FUNCTION_BLOCK TimerServer (* Updates time upon every REQ event and can be used to request time remotely. *)
  (* Standard: 61499-2 *)
  (* Version 1.0, 2017-09-05, Marc Jakobi, HTW Berlin *)
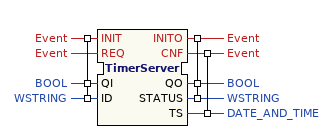
  EVENT_INPUT
    INIT WITH QI, ID; (* Initialization Request *)
    REQ; (* Service Request Event *)
  END_EVENT
  EVENT_OUTPUT
    INITO WITH QO, STATUS; (* Initialization Confirm *)
    CNF WITH TS; (* Service Indication *)
  END_EVENT
  VAR_INPUT
    QI : BOOL; (* Input event qualifier *)
    ID : WSTRING; (* Connection identifier *)
  END_VAR
  VAR_OUTPUT
    QO : BOOL; (* Output event qualifier *)
    STATUS : WSTRING; (* Service status *)
    TS : DATE_AND_TIME; (* Time stamp *)
  END_VAR
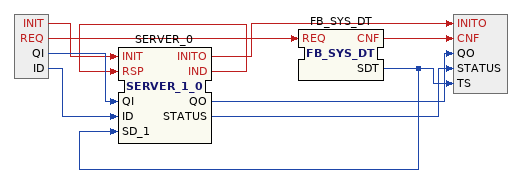
  FBS
    FB_SYS_DT : FB_SYS_DT;
    SERVER_0 : SERVER_1_0;
  END_FBS
  EVENT_CONNECTIONS
    FB_SYS_DT.CNF TO CNF;
    INIT TO SERVER_0.INIT;
    SERVER_0.INITO TO INITO;
    REQ TO FB_SYS_DT.REQ;
    SERVER_0.IND TO SERVER_0.RSP;
  END_CONNECTIONS
  DATA_CONNECTIONS
    FB_SYS_DT.SDT TO TS;
    QI TO SERVER_0.QI;
    ID TO SERVER_0.ID;
    SERVER_0.QO TO QO;
    SERVER_0.STATUS TO STATUS;
    FB_SYS_DT.SDT TO SERVER_0.SD_1;
  END_CONNECTIONS
END_FUNCTION_BLOCK
